FUNCTION_BLOCK T_ModuleCollectionNotifyModeChangedSuccess EXTENDS T_UnitTestBase
VAR
  list : T_SubModuleCollection;
  newModule, newModule2 : T_SubModuleMock; 
  actual1, actual2 : BOOL;
END_VAR

// Arrange
list.AddModule(newModule);
list.AddModule(newModule2);

//Act
list.NotifyModeChanged(E_PMLUnitMode.ePMLUnitMode_Maintenance);

//Assert
actual1 := newModule._newMode= E_PMLUnitMode.ePMLUnitMode_Maintenance;
actual2 := newModule2._newMode = E_PMLUnitMode.ePMLUnitMode_Maintenance;

assertion.AssertEquals_BOOL(TRUE, actual1, 'newModule._newState = E_PMLUnitMode.ePMLUnitMode_Maintenance');
assertion.AssertEquals_BOOL(TRUE, actual2, 'newModule2._newState = E_PMLUnitMode.ePMLUnitMode_Maintenance');
TestFinished();

END_FUNCTION_BLOCK

(* stored: Version 1.1.0.1, ProductVersion 3.1.4024.12
   POU T_ModuleCollectionNotifyModeChangedSuccess: Id {2fc17c18-8e96-40d4-9dfb-383b2a6945ae}, SpecialFunc None *)
